FUNCTION_BLOCK FT_AVG_200
VAR_INPUT
	IN : REAL;
	E : BOOL := TRUE;
	N : INT := 200;
	RST : BOOL;
END_VAR
VAR_OUTPUT
	AVG : REAL;
END_VAR
VAR
	buff : DELAY_200;
	i: INT;
	init : BOOL;
END_VAR

buff.N := LIMIT(0, N, 200);

IF NOT init OR rst THEN
	FOR i := 1 TO N DO
		buff(in := in);
	END_FOR;
	avg := in;
	init := TRUE;
ELSIF E THEN
	buff(in := in);
	avg := avg + (in - buff.out ) / INT_TO_REAL(N);
END_IF;

END_FUNCTION_BLOCK

(* stored: Version 1.1.0.1, ProductVersion 3.1.4024.3
   POU FT_AVG_200: Id {d89de838-a4ef-4478-9803-d954c8b7d37c}, SpecialFunc None *)
